{attribute 'pack_mode' := '2'}
TYPE ST_LIST_NODE_DATA :
STRUCT
  ProcessData     : ST_PROCESS_DATA;  // target data
END_STRUCT
END_TYPE

(* stored: Version 1.1.0.1, ProductVersion 3.1.4026.13
   DUT ST_LIST_NODE_DATA: Id {ef903480-c594-4df5-af23-86f29f792450} *)
